TYPE aS_AutoControl :
STRUCT
	Start: BOOL;
	Stop: BOOL;
	Setpoint: LREAL;
	ControlSignal: LREAL;
	Switch: BYTE;
END_STRUCT
END_TYPE

(* stored: Version 1.1.0.1, ProductVersion 3.1.4024.4
   DUT aS_AutoControl: Id {3778eaae-88e4-41c4-8e5f-afd374d3343a} *)
